// TwinCAT 3 PLC project ModbusServerTest
// ProgramVersion: 3.1.4023.0
// libraries:
//   Tc2_ModbusSrv, * (Beckhoff Automation GmbH)
//   Tc2_Standard, * (Beckhoff Automation GmbH)
//   Tc2_System, * (Beckhoff Automation GmbH)
//   Tc3_Module, * (Beckhoff Automation GmbH)
// project tree:
//   / PlcTask.TcTTO
//   POUs/ MAIN.TcPOU
// real-time tasks:
//   TASK PlcTask: cycle T#10ms, priority 20, ADS port 350
// I/O:
//   DEVICE Device 1 (EtherCAT Automation Protocol), AmsNetId 5.17.12.20.2.1
//   DEVICE Device 2 (EtherCAT Automation Protocol), AmsNetId 5.17.12.20.3.1

CONFIGURATION ModbusServerTest
    RESOURCE PLC ON TwinCAT3
        TASK PlcTask(INTERVAL := T#10ms, PRIORITY := 20);
        PROGRAM MAIN WITH PlcTask : MAIN;
    END_RESOURCE
END_CONFIGURATION

// ---- POUs/MAIN.TcPOU
PROGRAM MAIN
VAR
	sIpAddr : STRING[15] := '192.168.001.252';
	nport : UINT := 502;
	nUnitID : BYTE := 1;
	tTimeOut : TIME := T#1S;
	nOfReg : UINT := 10;
	nAddr :WORD := 0;
	
	fb_MBReadRegister: FB_MBReadRegs;
	bReadEnable: BOOL;
	bReadBusyFlag: BOOL;
	bReadErrorFlag: BOOL;
	nReadErrorID: UDINT;
	ireadReg : ARRAY[1..10] OF WORD;
	
	n :INT := 0;
	
	bWriteBusyFlag: BOOL;
	bWriteEnable: BOOL;
	fb_MBWriteRegister: FB_MBWriteRegs;
	bWriteErrorFlag: BOOL;
	nWriteErrorID: UDINT;
	iWriteReg : ARRAY[1..10] OF WORD;

END_VAR

(* Version history: 
Date          | Version    | created under        | Author          | Remark 
---------------------------------------------------------------------------------------- 
20/06/2022    | 1.0.0      | V3.1 (Build 4024.29) | Gokul G         | first release 
	* Basic Modbus TCP/IP Register Read/Write 
	
*) 
(* Modbus TCP/IP Communication  
1.First Install TF6250 Software in both Target & Enginnering PC Add Tc2_ModbusSrv Library 
2.In Main Program
	Variable 
	sIpAddr : STRING[15] := '192.168.001.252';
	nport : UINT := 502;
	nUnitID : BYTE := 1;
	tTimeOut : TIME := T#1S;
	nOfReg : UINT := 10;
	nAddr :WORD := 0;
	
	fb_MBReadRegister: FB_MBReadRegs;
	bReadEnable: BOOL;
	bReadBusyFlag: BOOL;
	bReadErrorFlag: BOOL;
	nReadErrorID: UDINT;
	ireadReg : ARRAY[1..10] OF WORD;
	
	n :INT := 0;
	
	bWriteBusyFlag: BOOL;
	bWriteEnable: BOOL;
	fb_MBWriteRegister: FB_MBWriteRegs;
	bWriteErrorFlag: BOOL;
	nWriteErrorID: UDINT;
	iWriteReg : ARRAY[1..10] OF WORD;
	
	Program 
	(* For Alternate Read & Write of Register *)
	IF n >= 100 AND NOT bReadBusyFlag THEN
		bReadEnable := TRUE;
	ELSIF n >= 200 AND NOT bWriteBusyFlag THEN
		bWriteEnable := TRUE;
		n := 0;
	END_IF
	n := n+1;

	(* Read Register *)
	fb_MBReadRegister(
		sIPAddr:= sIpAddr, 
		nTCPPort:= nport,
		nUnitID:= nUnitID, 
		nQuantity:= nOfReg , 
		nMBAddr:= nAddr , 
		cbLength:= SIZEOF(ireadReg), 
		pDestAddr:=ADR(ireadReg) , 
		bExecute:=bReadEnable , 
		tTimeout:= tTimeOut , 
		bBusy=> bReadBusyFlag, 
		bError=> bReadErrorFlag , 
		nErrId=> nReadErrorID , 
		cbRead=> );
	bReadEnable := FALSE;
	
	(* Write Register *)
	fb_MBWriteRegister(
		sIPAddr:= sIpAddr, 
		nTCPPort:= nport , 
		nUnitID:= nUnitID , 
		nQuantity:= nOfReg, 
		nMBAddr:= nAddr + 10 , 
		cbLength:= SIZEOF(iWriteReg), 
		pSrcAddr:= ADR(iWriteReg), 
		bExecute:= bWriteEnable, 
		tTimeout:= tTimeOut, 
		bBusy=> bWriteBusyFlag, 
		bError=> bWriteErrorFlag, 
		nErrId=> nWriteErrorID );	
	bWriteEnable := FALSE;
3.Set IP Adress of Servers as per requirement & port should be specified (Usally 502 but it can be changed if multiple modbus servers are there in same IP)
4.Program will alternately read & write register every 1 secs

Note :
	If Address in Modscan is 1 then in MBAddress it should be 0 (-1)
	
*)

(* For Alternate Read & Write of Register *)
IF n >= 100 AND NOT bReadBusyFlag THEN
	bReadEnable := TRUE;
ELSIF n >= 200 AND NOT bWriteBusyFlag THEN
	bWriteEnable := TRUE;
	n := 0;
END_IF
n := n+1;

(* Read Register *)
fb_MBReadRegister(
	sIPAddr:= sIpAddr, 
	nTCPPort:= nport,
	nUnitID:= nUnitID, 
	nQuantity:= nOfReg , 
	nMBAddr:= nAddr , 
	cbLength:= SIZEOF(ireadReg), 
	pDestAddr:=ADR(ireadReg) , 
	bExecute:=bReadEnable , 
	tTimeout:= tTimeOut , 
	bBusy=> bReadBusyFlag, 
	bError=> bReadErrorFlag , 
	nErrId=> nReadErrorID , 
	cbRead=> );
bReadEnable := FALSE;

(* Write Register *)
fb_MBWriteRegister(
	sIPAddr:= sIpAddr, 
	nTCPPort:= nport , 
	nUnitID:= nUnitID , 
	nQuantity:= nOfReg, 
	nMBAddr:= nAddr + 10 , 
	cbLength:= SIZEOF(iWriteReg), 
	pSrcAddr:= ADR(iWriteReg), 
	bExecute:= bWriteEnable, 
	tTimeout:= tTimeOut, 
	bBusy=> bWriteBusyFlag, 
	bError=> bWriteErrorFlag, 
	nErrId=> nWriteErrorID );	
bWriteEnable := FALSE;

END_PROGRAM
